Yaskawa INFORM job: R1_W9_MP.JBI

/JOB
//NAME R1_W9_MP
///FOLDERNAME INNE
//POS
///NPOS 101,101,101,5,0,0
///TOOL 0
///POSTYPE PULSE
///PULSE
C00000=-93820,47590,81922,-44796,65389,-14940
C00001=-93822,47583,81914,-44796,65389,-14941
C00002=-93823,47580,81910,-44796,65389,-14942
C00003=-93824,47578,81909,-44796,65389,-14942
C00004=-93823,47580,81910,-44796,65389,-14942
C00005=-93828,47581,81911,-54669,68995,-12236
C00006=-93828,47578,81908,-54669,68995,-12236
C00007=-93828,47581,81911,-54669,68995,-12236
C00008=-93312,45364,79055,-34090,63475,-18022
C00009=-93821,47567,81895,-34291,62777,-17990
C00010=-93258,45661,79407,-34104,63441,-17988
C00011=-93819,47569,81898,-34292,62777,-17990
C00012=-93817,47575,81906,-34292,62777,-17989
C00013=-93817,47575,81906,-34292,62777,21711
C00014=-93810,47570,81900,-15066,61616,44422
C00015=-93811,47561,81889,-15066,61617,44422
C00016=-93812,47557,81884,-15065,61618,44421
C00017=-93814,47558,81885,-15065,61617,44421
C00018=-93814,47555,81882,-15065,61618,44421
C00019=-93814,47558,81885,-15065,61617,44421
C00020=-93812,47557,81884,-15065,61618,44421
C00021=-92182,50271,85003,-15131,61382,45028
C00022=-93813,47553,81880,-15065,61618,44421
C00023=-92198,50243,84970,-15130,61385,45022
C00024=-93812,47557,81884,-15065,61618,44421
C00025=-93816,47564,81892,-25041,56991,45512
C00026=-93816,47564,81892,-25041,56991,45512
C00027=-93816,47564,81892,-25041,56991,45512
C00028=-93817,47563,81891,-25041,56991,45512
C00029=-93816,47566,81895,-25041,56991,45512
C00030=-93815,47576,81906,-25042,56989,45513
C00031=-93816,47549,81875,-44212,47727,7509
C00032=-93817,47544,81870,-44212,47727,7508
C00033=-93818,47542,81867,-44211,47727,7508
C00034=-93817,47537,81861,-44211,47728,7507
C00035=-93818,47535,81859,-44210,47728,7507
C00036=-93817,47537,81861,-44211,47728,7507
C00037=-93818,47542,81867,-44211,47727,7508
C00038=-94360,44479,77062,-43304,48500,6770
C00039=-93819,47539,81864,-44211,47727,7507
C00040=-94433,44095,76454,-43190,48598,6676
C00041=-93818,47542,81867,-44211,47727,7508
C00042=-93818,47542,81867,-44211,47727,7508
C00043=-93817,47539,81864,-44211,47728,7507
C00044=-93817,47539,81864,-44211,47728,7507
C00045=-93817,47539,81864,-44211,47728,7507
C00046=-93818,47544,81869,-44212,47727,7508
C00047=-93818,47544,81869,-44212,47727,7508
C00048=-93817,47544,81870,-44212,47727,7508
C00049=-93816,47549,81875,-44212,47727,7509
C00050=-93808,47528,81852,-36012,54490,-21231
C00051=-93810,47523,81845,-36011,54490,-21232
C00052=-93811,47521,81843,-36011,54490,-21232
C00053=-93812,47519,81841,-36011,54490,-21233
C00054=-93811,47521,81843,-36011,54490,-21232
C00055=-93811,47521,81843,-36011,54490,-21232
C00056=-93811,47521,81843,-36011,54490,-21232
C00057=-93811,47521,81843,-36011,54490,-21232
C00058=-93811,47525,81848,-36011,54490,-21232
C00059=-93808,47531,81854,-36012,54490,-21231
C00060=-92781,31963,61007,-34275,58868,-22415
C00061=-147445,47546,81835,-34359,45417,-40791
C00062=-149267,32865,67814,-33397,45672,-41812
C00063=-140416,53932,103867,-53063,49753,-24186
C00064=-140498,61069,114440,-55068,47999,-22830
C00065=-140379,61139,114538,-55063,48040,-22793
C00066=-141057,43414,93234,-54762,45840,-22344
C00067=-141971,41882,92369,-54635,45639,-23532
C00068=-141612,43108,94051,-55498,44972,-21992
C00069=-141612,44298,95907,-55937,44664,-21713
C00070=-141537,44510,96728,-56259,44468,-21485
C00071=-139753,46250,105668,-60066,42792,-18577
C00072=-139544,42960,101093,-58991,43483,-19175
C00073=-139488,29243,80111,-54132,46852,-22269
C00074=-147382,25464,47554,-24500,64095,-34288
C00075=-147526,44634,78086,-43145,44718,-41029
C00076=-134037,47519,81818,-10606,38218,-38188
C00077=-134048,47518,81817,-10600,38217,-38193
C00078=-134051,47520,81819,-10599,38217,-38194
C00079=-134052,47520,81820,-10599,38216,-38195
C00080=-134598,47405,82622,-10458,37608,-38382
C00081=-134154,43284,75981,-10234,39599,-38425
C00082=-134052,47525,81825,-10599,38215,-38195
C00083=-134052,47525,81825,-10599,38215,-38195
C00084=-134053,47530,81831,-10598,38214,-38195
C00085=-134052,47530,81831,-10599,38215,-38195
C00086=-134050,47528,81829,-10600,38215,-38193
C00087=-134038,47529,81829,-10605,38216,-38188
C00088=-107226,47597,81926,-62456,56100,-14962
C00089=-107237,47581,81907,-62455,56095,-14965
C00090=-107238,47574,81900,-62455,56095,-14966
C00091=-107239,47572,81897,-62455,56095,-14966
C00092=-107128,43336,76056,-61624,56853,-15625
C00093=-107129,47038,82405,-62787,55875,-14663
C00094=-107239,47566,81891,-62454,56095,-14967
C00095=-107238,47552,81874,-62452,56097,-14968
C00096=-107238,47547,81869,-62452,56097,-14968
C00097=-107240,47545,81866,-68624,54366,-16050
C00098=-107240,47547,81869,-68624,54366,-16049
C00099=-107238,47554,81876,-68625,54367,-16048
C00100=-107228,47571,81895,-68625,54372,-16045
BC00000=250791,53675,753741
BC00001=248916,56711,729871
BC00002=248167,57926,720323
BC00003=248155,59571,714678
BC00004=248167,57926,720323
BC00005=258176,50768,676178
BC00006=256129,49929,673230
BC00007=258176,50768,676178
BC00008=232157,60047,738004
BC00009=233389,58670,733055
BC00010=232157,60047,738004
BC00011=232431,59052,748136
BC00012=233115,56565,773466
BC00013=233115,56565,773466
BC00014=214797,73994,838742
BC00015=210542,75620,816743
BC00016=208839,76270,807943
BC00017=213516,76274,789192
BC00018=211688,76276,783998
BC00019=213516,76274,789192
BC00020=208839,76270,807943
BC00021=205362,76890,805337
BC00022=208439,76892,792997
BC00023=205362,76890,805337
BC00024=208839,76270,807943
BC00025=221278,65723,777613
BC00026=221279,70331,777630
BC00027=221278,65723,777613
BC00028=222479,60892,767842
BC00029=224368,59825,775652
BC00030=229092,57156,795177
BC00031=210723,30242,763895
BC00032=209625,36131,747039
BC00033=209185,38486,740297
BC00034=204260,38488,740270
BC00035=204264,38490,732205
BC00036=204260,38488,740270
BC00037=209185,38486,740297
BC00038=210873,38455,729592
BC00039=208484,38456,729579
BC00040=210873,38455,729592
BC00041=209185,38486,740297
BC00042=210869,40530,740313
BC00043=205997,40531,742232
BC00044=205998,42836,742240
BC00045=205997,40531,742232
BC00046=210869,40530,740313
BC00047=209185,38486,740297
BC00048=209625,36131,747039
BC00049=210723,30242,763895
BC00050=180235,54254,818576
BC00051=180221,57233,793797
BC00052=180216,58425,783885
BC00053=180220,58427,775820
BC00054=180216,58425,783885
BC00055=182182,60992,784445
BC00056=182163,63296,784453
BC00057=182182,60992,784445
BC00058=182188,59800,794356
BC00059=182201,56821,819136
BC00060=245303,56821,1001710
BC00061=376901,73323,906143
BC00062=376826,95199,858168
BC00063=371848,95135,813088
BC00064=371848,95135,813088
BC00065=371848,95135,813088
BC00066=371848,95135,813088
BC00067=371848,95135,813088
BC00068=371848,95135,813088
BC00069=371848,95135,813088
BC00070=371848,95135,813088
BC00071=371849,95134,813085
BC00072=371849,95134,813085
BC00073=371849,95134,813085
BC00074=371849,95134,892955
BC00075=397580,75248,898673
BC00076=291745,42722,928164
BC00077=291796,42753,820630
BC00078=293348,46102,797011
BC00079=293969,47442,787564
BC00080=293969,47442,787564
BC00081=293969,47442,787564
BC00082=297987,45710,781283
BC00083=298996,45275,779706
BC00084=303015,43543,773425
BC00085=302394,42203,782873
BC00086=300841,38854,806491
BC00087=300790,38822,914026
BC00088=276425,36483,823377
BC00089=276476,36514,715843
BC00090=273728,40692,695282
BC00091=272628,42364,687058
BC00092=272628,42364,687058
BC00093=272628,42364,687058
BC00094=267850,42326,687032
BC00095=255369,42226,686964
BC00096=250793,42190,686939
BC00097=252133,35730,663831
BC00098=253294,33956,671687
BC00099=256197,29521,691326
BC00100=256146,29489,798860
EC00000=-798156,-556475
EC00001=-798156,-556475
EC00002=-798156,-556475
EC00003=-798156,-556475
EC00004=-798156,-556475
EC00005=-798156,-556475
EC00006=-798156,-556475
EC00007=-798156,-556475
EC00008=-798156,-556475
EC00009=-798156,-556475
EC00010=-798156,-556475
EC00011=-798156,-556475
EC00012=-798156,-556475
EC00013=-798156,-556475
EC00014=-798156,-556475
EC00015=-798156,-556475
EC00016=-798156,-556475
EC00017=-798156,-556475
EC00018=-798156,-556475
EC00019=-798156,-556475
EC00020=-798156,-556475
EC00021=-798156,-556475
EC00022=-798156,-556475
EC00023=-798156,-556475
EC00024=-798156,-556475
EC00025=-798156,-556475
EC00026=-798156,-556475
EC00027=-798156,-556475
EC00028=-798156,-556475
EC00029=-798156,-556475
EC00030=-798156,-556475
EC00031=-798156,-556475
EC00032=-798156,-556475
EC00033=-798156,-556475
EC00034=-798156,-556475
EC00035=-798156,-556475
EC00036=-798156,-556475
EC00037=-798156,-556475
EC00038=-798156,-556475
EC00039=-798156,-556475
EC00040=-798156,-556475
EC00041=-798156,-556475
EC00042=-798156,-556475
EC00043=-798156,-556475
EC00044=-798156,-556475
EC00045=-798156,-556475
EC00046=-798156,-556475
EC00047=-798156,-556475
EC00048=-798156,-556475
EC00049=-798156,-556475
EC00050=-798156,-556475
EC00051=-798156,-556475
EC00052=-798156,-556475
EC00053=-798156,-556475
EC00054=-798156,-556475
EC00055=-798156,-556475
EC00056=-798156,-556475
EC00057=-798156,-556475
EC00058=-798156,-556475
EC00059=-798156,-556475
EC00060=-798156,-556475
EC00061=-798156,-556475
EC00062=-798154,-556474
EC00063=-798154,-556474
EC00064=-798154,-556474
EC00065=-798154,-556474
EC00066=-798154,-556474
EC00067=-798154,-556474
EC00068=-798154,-556474
EC00069=-798154,-556474
EC00070=-798154,-556474
EC00071=-798153,-556474
EC00072=-798153,-556474
EC00073=-798153,-556474
EC00074=-798153,-556474
EC00075=-798156,-556475
EC00076=-798156,-556475
EC00077=-798156,-556475
EC00078=-798156,-556475
EC00079=-798156,-556475
EC00080=-798156,-556475
EC00081=-798156,-556475
EC00082=-798156,-556475
EC00083=-798156,-556475
EC00084=-798156,-556475
EC00085=-798156,-556475
EC00086=-798156,-556475
EC00087=-798156,-556475
EC00088=-798156,-556475
EC00089=-798156,-556475
EC00090=-798156,-556475
EC00091=-798156,-556475
EC00092=-798156,-556475
EC00093=-798156,-556475
EC00094=-798156,-556475
EC00095=-798156,-556475
EC00096=-798156,-556475
EC00097=-798156,-556475
EC00098=-798156,-556475
EC00099=-798156,-556475
EC00100=-798156,-556475
///POSTYPE BASE
///RECTAN
///RCONF 0,0,0,0,1,0,0,0,0,0,0,0,0,0,0,0,0,0,0,0,0,0,0,0
P00006=2.006,1.622,-0.565,0.0000,0.0000,0.0000
P00021=0.073,2.058,-0.109,0.0000,0.0000,0.0000
P00022=2.006,1.622,-0.565,0.0000,0.0000,0.0000
///RCONF 0,0,0,0,0,0,0,0,0,0,0,0,0,0,0,0,0,0,0,0,0,0,0,0
P00023=-2.957,-4.083,2.762,0.0000,0.0000,0.0000
P00024=-1.466,-0.226,-0.419,0.0000,0.0000,0.0000
//INST
///DATE 2023/10/04 16:41
///ATTR SC,RW
///GROUP1 RB1,BS1
///GROUP2 ST1
NOP
'r1_W9
'Path S790 (for W407)
SSFTOF
MOVL C00000 BC00000 V=1000.0  +MOVJ EC00000 VJ=100.00
MOVL C00001 BC00001 V=400.0  +MOVJ EC00001 VJ=100.00
SMOVL C00002 BC00002 V=60.0  +MOVJ EC00002
SREFP 3 C00003 BC00003  +REFP EC00003
CALL JOB:SEARCH-R1-S1
SET P021 P006
SSFTON P021
SMOVL C00004 BC00004 V=60.0  +MOVJ EC00004
SMOVL C00005 BC00005 V=60.0  +MOVJ EC00005
SREFP 3 C00006 BC00006  +REFP EC00006
CALL JOB:SEARCH-R1-S1
SET P021 P006
SSFTON P021
SMOVL C00007 BC00007 V=60.0  +MOVJ EC00007
SMOVL C00008 BC00008 V=60.0  +MOVJ EC00008
SREFP 3 C00009 BC00009  +REFP EC00009
CALL JOB:SEARCH-R1-S1
SET P021 P006
SSFTON P021
SMOVL C00010 BC00010 V=60.0  +MOVJ EC00010
MOVL C00011 BC00011 V=400.0  +MOVJ EC00011 VJ=100.00
MOVL C00012 BC00012 V=1000.0  +MOVJ EC00012 VJ=100.00
'Path S791 (for W407)
MOVL C00013 BC00013 V=1000.0  +MOVJ EC00013 VJ=100.00
MOVL C00014 BC00014 V=1000.0  +MOVJ EC00014 VJ=100.00
MOVL C00015 BC00015 V=400.0  +MOVJ EC00015 VJ=100.00
SMOVL C00016 BC00016 V=100.0  +MOVJ EC00016
SMOVL C00017 BC00017 V=60.0  +MOVJ EC00017
SREFP 3 C00018 BC00018  +REFP EC00018
CALL JOB:SEARCH-R1-S1
SET P022 P006
SSFTON P022
SMOVL C00019 BC00019 V=60.0  +MOVJ EC00019
SMOVL C00020 BC00020 V=100.0  +MOVJ EC00020
SMOVL C00021 BC00021 V=60.0  +MOVJ EC00021
SREFP 3 C00022 BC00022  +REFP EC00022
CALL JOB:SEARCH-R1-S1
SET P022 P006
SSFTON P022
SMOVL C00023 BC00023 V=60.0  +MOVJ EC00023
SMOVL C00024 BC00024 V=100.0  +MOVJ EC00024
SMOVL C00025 BC00025 V=60.0  +MOVJ EC00025
SREFP 3 C00026 BC00026  +REFP EC00026
CALL JOB:SEARCH-R1-S1
SET P022 P006
SSFTON P022
SMOVL C00027 BC00027 V=60.0  +MOVJ EC00027
SMOVL C00028 BC00028 V=100.0  +MOVJ EC00028
MOVL C00029 BC00029 V=400.0  +MOVJ EC00029 VJ=100.00
MOVL C00030 BC00030 V=1000.0  +MOVJ EC00030 VJ=100.00
'Path S802 (for W408)
SSFTOF
MOVL C00031 BC00031 V=1000.0  +MOVJ EC00031 VJ=100.00
MOVL C00032 BC00032 V=400.0  +MOVJ EC00032 VJ=100.00
SMOVL C00033 BC00033 V=100.0  +MOVJ EC00033
SMOVL C00034 BC00034 V=60.0  +MOVJ EC00034
SREFP 3 C00035 BC00035  +REFP EC00035
CALL JOB:SEARCH-R1-S1
SET P023 P006
SSFTON P023
SMOVL C00036 BC00036 V=60.0  +MOVJ EC00036
SMOVL C00037 BC00037 V=100.0  +MOVJ EC00037
SMOVL C00038 BC00038 V=60.0  +MOVJ EC00038
SREFP 3 C00039 BC00039  +REFP EC00039
CALL JOB:SEARCH-R1-S1
SET P023 P006
SSFTON P023
SMOVL C00040 BC00040 V=60.0  +MOVJ EC00040
SMOVL C00041 BC00041 V=100.0  +MOVJ EC00041
SMOVL C00042 BC00042 V=100.0  +MOVJ EC00042
SMOVL C00043 BC00043 V=60.0  +MOVJ EC00043
SREFP 3 C00044 BC00044  +REFP EC00044
CALL JOB:SEARCH-R1-S1
SET P023 P006
SSFTON P023
SMOVL C00045 BC00045 V=60.0  +MOVJ EC00045
SMOVL C00046 BC00046 V=100.0  +MOVJ EC00046
SMOVL C00047 BC00047 V=100.0  +MOVJ EC00047
MOVL C00048 BC00048 V=400.0  +MOVJ EC00048 VJ=100.00
MOVL C00049 BC00049 V=1000.0  +MOVJ EC00049 VJ=100.00
'Path S803 (for W408)
SSFTOF
MOVL C00050 BC00050 V=1000.0  +MOVJ EC00050 VJ=100.00
MOVL C00051 BC00051 V=400.0  +MOVJ EC00051 VJ=100.00
SMOVL C00052 BC00052 V=60.0  +MOVJ EC00052
SREFP 3 C00053 BC00053  +REFP EC00053
CALL JOB:SEARCH-R1-S1
SET P024 P006
SSFTON P024
SMOVL C00054 BC00054 V=60.0  +MOVJ EC00054
SMOVL C00055 BC00055 V=60.0  +MOVJ EC00055
SREFP 3 C00056 BC00056  +REFP EC00056
CALL JOB:SEARCH-R1-S1
SET P024 P006
SSFTON P024
SMOVL C00057 BC00057 V=60.0  +MOVJ EC00057
MOVL C00058 BC00058 V=400.0  +MOVJ EC00058 VJ=100.00
MOVL C00059 BC00059 V=1000.0  +MOVJ EC00059 VJ=100.00
'Path W407
SSFTOF
MOVJ C00060 BC00060 VJ=100.00  +MOVJ EC00060 VJ=100.00
MOVJ C00061 BC00061 VJ=100.00  +MOVJ EC00061 VJ=100.00
MOVJ C00062 BC00062 VJ=100.00  +MOVJ EC00062 VJ=100.00
MOVJ C00063 BC00063 VJ=100.00  +MOVJ EC00063 VJ=100.00
SSFTON P022
SMOVL C00064 BC00064 V=400.0  +MOVJ EC00064
SMOVL C00065 BC00065 V=100.0 PL=0  +MOVJ EC00065
SREFP 1 C00066 BC00066  +REFP EC00066
SREFP 2 C00067 BC00067  +REFP EC00067
MACRO1 MJ#(0) ARGF0
ARCON
SMOVL C00068 BC00068 V=10.0  +MOVJ EC00068
SMOVL C00069 BC00069 V=10.0  +MOVJ EC00069
SMOVL C00070 BC00070 V=10.0  +MOVJ EC00070
SSFTON P021
SMOVL C00071 BC00071 V=10.0  +MOVJ EC00071
SMOVL C00072 BC00072 V=10.0  +MOVJ EC00072
ARCOF
SMOVL C00073 BC00073 V=400.0  +MOVJ EC00073
SMOVL C00074 BC00074 V=1000.0  +MOVJ EC00074
SMOVL C00075 BC00075 V=1000.0  +MOVJ EC00075
SSFTOF
'Path W408
SSFTOF
MOVJ C00076 BC00076 VJ=100.00  +MOVJ EC00076 VJ=100.00
SSFTON P023
SMOVL C00077 BC00077 V=1000.0  +MOVJ EC00077
SMOVL C00078 BC00078 V=400.0  +MOVJ EC00078
SMOVL C00079 BC00079 V=100.0 PL=0  +MOVJ EC00079
SREFP 1 C00080 BC00080  +REFP EC00080
SREFP 2 C00081 BC00081  +REFP EC00081
MACRO1 MJ#(0) ARGF0
ARCON
SMOVL C00082 BC00082 V=10.0  +MOVJ EC00082
SSFTON P022
SMOVL C00083 BC00083 V=10.0  +MOVJ EC00083
SMOVL C00084 BC00084 V=10.0  +MOVJ EC00084
ARCOF
SMOVL C00085 BC00085 V=400.0  +MOVJ EC00085
SMOVL C00086 BC00086 V=1000.0  +MOVJ EC00086
SMOVL C00087 BC00087 V=1000.0  +MOVJ EC00087
SSFTOF
'Path W409
SSFTOF
MOVJ C00088 BC00088 VJ=100.00  +MOVJ EC00088 VJ=100.00
SSFTON P023
SMOVL C00089 BC00089 V=1000.0  +MOVJ EC00089
SMOVL C00090 BC00090 V=400.0  +MOVJ EC00090
SMOVL C00091 BC00091 V=100.0 PL=0  +MOVJ EC00091
SREFP 1 C00092 BC00092  +REFP EC00092
SREFP 2 C00093 BC00093  +REFP EC00093
MACRO1 MJ#(0) ARGF0
ARCON
SMOVL C00094 BC00094 V=10.0  +MOVJ EC00094
SSFTON P024
SMOVL C00095 BC00095 V=10.0  +MOVJ EC00095
SMOVL C00096 BC00096 V=10.0  +MOVJ EC00096
SMOVL C00097 BC00097 V=10.0  +MOVJ EC00097
ARCOF
SMOVL C00098 BC00098 V=400.0  +MOVJ EC00098
SMOVL C00099 BC00099 V=1000.0  +MOVJ EC00099
SMOVL C00100 BC00100 V=1000.0  +MOVJ EC00100
SSFTOF
END
